GLOBALCONSTANTS modbus_const (* Global constants *)
  (* Standard: 61499-1 *)
  (* Version 1.0, 2024-08-18, franz *)
  VAR_GLOBAL CONSTANT
    ID_01_RTU : WSTRING := "modbus[rtu:/dev/uart/1:9600:N:8:1:delay:1:500:c0..7:c0..7]";
    ID_01_TCP : WSTRING := "modbus[tcp:192.168.1.99:502:1:500:h468:h470]";
    ID_02_TCP : WSTRING := "modbus[tcp:192.168.1.99:502:1:500:h51:]";
  END_VAR
END_GLOBALCONSTANTS
